# EPICS autosave request: utcaApp/Db/bpm_common.req
file "trigger_iface.req", P=${P}, R=${R}, TRIGGER_NAME=TRIGGER
file "orbit_intlk.req", P=${P}, R=${R}

file "bpm_common_single.req", P=${P1}, R=${R1}
file "bpm_common_single.req", P=${P2}, R=${R2}
